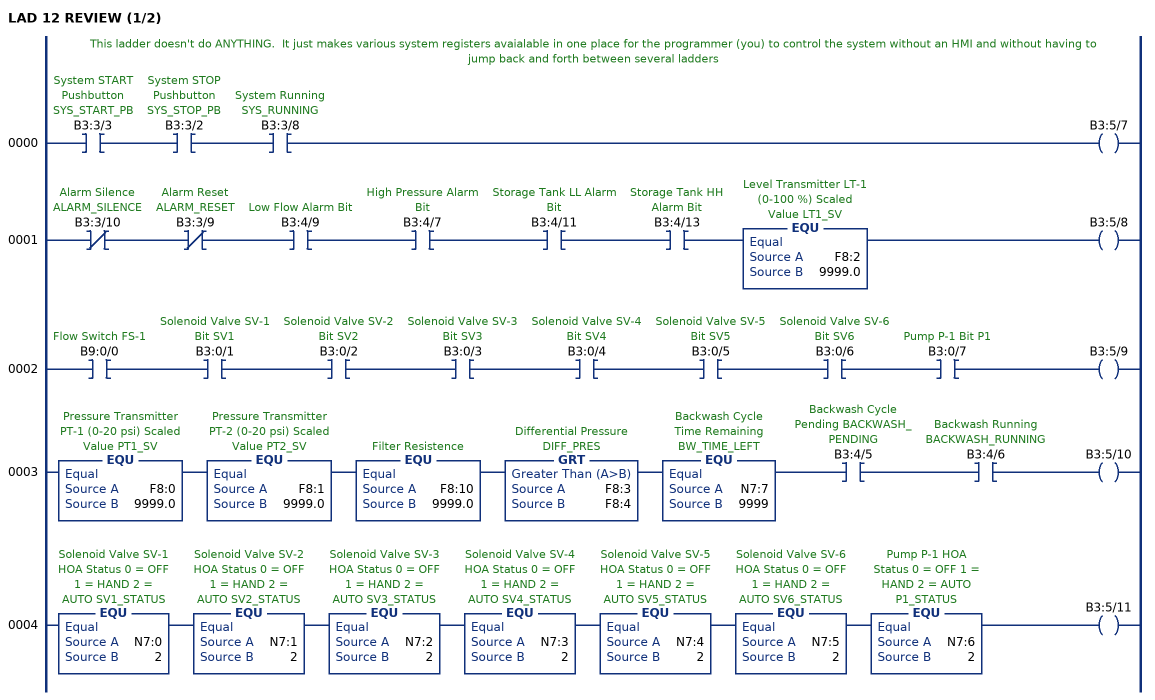
% Rung: 0 %
% This ladder doesn't do ANYTHING.  It just makes various system registers avaialable in one place for the programmer (you) to control the system without an HMI and without having to jump back and forth between several ladders %
SOR XIC B3:3/3 XIC B3:3/2 XIC B3:3/8 OTE B3:5/7 EOR
%   B3:3/3  SYS_START_PB  "System START Pushbutton" %
%   B3:3/2  SYS_STOP_PB  "System STOP Pushbutton" %
%   B3:3/8  SYS_RUNNING  "System Running" %
% Rung: 1 %
SOR XIO B3:3/10 XIO B3:3/9 XIC B3:4/9 XIC B3:4/7 XIC B3:4/11 XIC B3:4/13 EQU F8:2 9999.0 OTE B3:5/8 EOR
%   B3:3/10  ALARM_SILENCE  "Alarm Silence" %
%   B3:3/9  ALARM_RESET  "Alarm Reset" %
%   B3:4/9  "Low Flow Alarm Bit" %
%   B3:4/7  "High Pressure Alarm Bit" %
%   B3:4/11  "Storage Tank LL Alarm Bit" %
%   B3:4/13  "Storage Tank HH Alarm Bit" %
%   F8:2  LT1_SV  "Level Transmitter LT-1 (0-100 %) Scaled Value" %
% Rung: 2 %
SOR XIC B9:0/0 XIC B3:0/1 XIC B3:0/2 XIC B3:0/3 XIC B3:0/4 XIC B3:0/5 XIC B3:0/6 XIC B3:0/7 OTE B3:5/9 EOR
%   B9:0/0  "Flow Switch FS-1" %
%   B3:0/1  SV1  "Solenoid Valve SV-1 Bit" %
%   B3:0/2  SV2  "Solenoid Valve SV-2 Bit" %
%   B3:0/3  SV3  "Solenoid Valve SV-3 Bit" %
%   B3:0/4  SV4  "Solenoid Valve SV-4 Bit" %
%   B3:0/5  SV5  "Solenoid Valve SV-5 Bit" %
%   B3:0/6  SV6  "Solenoid Valve SV-6 Bit" %
%   B3:0/7  P1  "Pump P-1 Bit" %
% Rung: 3 %
SOR EQU F8:0 9999.0 EQU F8:1 9999.0 EQU F8:10 9999.0 GRT F8:3 F8:4 EQU N7:7 9999 XIC B3:4/5 XIC B3:4/6 OTE B3:5/10 EOR
%   F8:0  PT1_SV  "Pressure Transmitter PT-1 (0-20 psi) Scaled Value" %
%   F8:1  PT2_SV  "Pressure Transmitter PT-2 (0-20 psi) Scaled Value" %
%   F8:10  "Filter Resistence" %
%   F8:3  DIFF_PRES  "Differential Pressure" %
%   F8:4  BACKWASH_SP  "Backwash Cycle Trigger Setpoint" %
%   N7:7  BW_TIME_LEFT  "Backwash Cycle Time Remaining" %
%   B3:4/5  BACKWASH_PENDING  "Backwash Cycle Pending" %
%   B3:4/6  BACKWASH_RUNNING  "Backwash Running" %
% Rung: 4 %
SOR EQU N7:0 2 EQU N7:1 2 EQU N7:2 2 EQU N7:3 2 EQU N7:4 2 EQU N7:5 2 EQU N7:6 2 OTE B3:5/11 EOR
%   N7:0  SV1_STATUS  "Solenoid Valve SV-1 HOA Status 0 = OFF 1 = HAND 2 = AUTO" %
%   N7:1  SV2_STATUS  "Solenoid Valve SV-2 HOA Status 0 = OFF 1 = HAND 2 = AUTO" %
%   N7:2  SV3_STATUS  "Solenoid Valve SV-3 HOA Status 0 = OFF 1 = HAND 2 = AUTO" %
%   N7:3  SV4_STATUS  "Solenoid Valve SV-4 HOA Status 0 = OFF 1 = HAND 2 = AUTO" %
%   N7:4  SV5_STATUS  "Solenoid Valve SV-5 HOA Status 0 = OFF 1 = HAND 2 = AUTO" %
%   N7:5  SV6_STATUS  "Solenoid Valve SV-6 HOA Status 0 = OFF 1 = HAND 2 = AUTO" %
%   N7:6  P1_STATUS  "Pump P-1 HOA Status 0 = OFF 1 = HAND 2 = AUTO" %

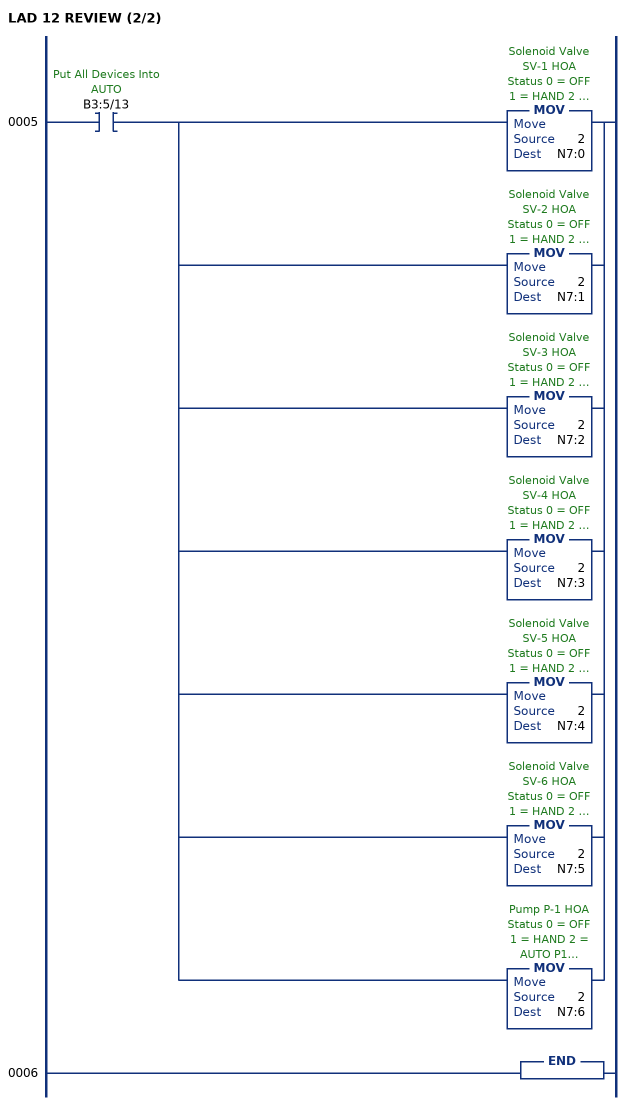
% Rung: 5 %
SOR XIC B3:5/13 BST MOV 2 N7:0 NXB MOV 2 N7:1 NXB MOV 2 N7:2 NXB MOV 2 N7:3 NXB MOV 2 N7:4 NXB MOV 2 N7:5 NXB MOV 2 N7:6 BND EOR
%   B3:5/13  "Put All Devices Into AUTO" %
%   N7:0  SV1_STATUS  "Solenoid Valve SV-1 HOA Status 0 = OFF 1 = HAND 2 = AUTO" %
%   N7:1  SV2_STATUS  "Solenoid Valve SV-2 HOA Status 0 = OFF 1 = HAND 2 = AUTO" %
%   N7:2  SV3_STATUS  "Solenoid Valve SV-3 HOA Status 0 = OFF 1 = HAND 2 = AUTO" %
%   N7:3  SV4_STATUS  "Solenoid Valve SV-4 HOA Status 0 = OFF 1 = HAND 2 = AUTO" %
%   N7:4  SV5_STATUS  "Solenoid Valve SV-5 HOA Status 0 = OFF 1 = HAND 2 = AUTO" %
%   N7:5  SV6_STATUS  "Solenoid Valve SV-6 HOA Status 0 = OFF 1 = HAND 2 = AUTO" %
%   N7:6  P1_STATUS  "Pump P-1 HOA Status 0 = OFF 1 = HAND 2 = AUTO" %
% Rung: 6 %
SOR END EOR

OTHER DOCUMENTED ADDRESSES
  DFILE:0  "OUTPUT"
  DFILE:1  "INPUT"
  DFILE:2  "STATUS"
  DFILE:3  "BINARY"
  DFILE:4  "TIMER"
  DFILE:5  "COUNTER"
  DFILE:6  "CONTROL"
  DFILE:7  "INTEGER"
  DFILE:8  "FLOAT"
  DFILE:9  "DIGITAL IO"
  DFILE:10  "ANALOG IO"

COMMENTS NOT ATTACHED TO A CURRENT RUNG
  T4:1: High Pressure alarm

DATA TABLE (non-zero values as saved)
DATA T4
% .PRE .ACC %
% T4:0 % 5 0
% T4:1 % 5 0
% T4:2 % 5 0
% T4:3 % 5 0
% T4:4 % 5 0
% T4:5 % 2 0
% T4:6 % 60 0
% T4:7 % 2 0
% T4:8 % 2 0
% T4:9 % 500 0
% T4:10 % 2 0
% T4:11 % 5 0
% T4:12 % 500 0
% T4:13 % 60 0
% T4:14 % 5 0
DATA F8
% F8:0 % 0 0 0 0 5
% F8:5 % 15 10 90 20 80
